// TIA Portal V19 export
VAR_GLOBAL   // PLC tag table "HU_Decoilers_IO"
   HU_Decoilers_Pump_C AT %Q0.6 : Bool;   // 660KA1
   HU_Decoilers_Pump_Fdbk AT %I3.1 : Bool;   // 660KM1
END_VAR
